/// This enumeration contains all steps that are used by the various sequences of a unit.
/// Sequences use a subrange (***Begin to ***End) of this enumeration.
{attribute 'qualified_only'}
{attribute 'to_string'}
TYPE HandlingStep :
(
  Undefined := 0
  
  ,BootBegin
  ,BootEnd 

  ,StopBegin
  ,StopEnd

  ,AutomaticBegin
  ,AutomaticSwitch
  ,AutomaticMoveInterpolatedVelocity
  ,AutomaticEnd
  
  ,GoHomeBegin
  ,GoHomeJoint3
  ,GoHomeJoint12
  ,GoHomeJoint2
  ,GoHomeEnd 
  
  ,FaultReactionBegin
  ,FaultReactionEnd
);
END_TYPE

(* stored: Version 1.1.0.1
   DUT HandlingStep: Id {7cd5c1c8-8bf6-476d-b1ec-c4d158904feb} *)
